{attribute addProperty BoxType "EL6851-0010-0019"}
{attribute addProperty Id "DMX_StatusAT %I*DMX_Status_A8F3522A6480DMX_Channel_1_64AT %I*DMX_Channel_D03720FB512640WcStateAT %I*WcState_98A4DF7520.250InfoDataAT %I*InfoData_BC63D37F80100"}
{attribute addProperty CRC "2912125561"}
{attribute addProperty SizeInBites "658"}
{attribute addProperty SizeInBytes "82.25"}
TYPE EL6851_20762A18 :
STRUCT
	{attribute addProperty Name "DMX_Status"}
	DMX_Status : DMX_Status_A8F3522A;
	{attribute addProperty Name "DMX_Channel_1_64"}
	DMX_Channel_1_64 : DMX_Channel_D03720FB;
	{attribute addProperty Name "WcState"}
	WcState : WcState_98A4DF75;
	{attribute addProperty Name "InfoData"}
	InfoData : InfoData_BC63D37F;
END_STRUCT
END_TYPE

(* stored: Version 1.2.0.0, ProductVersion 3.1.4024.9
   DUT EL6851_20762A18: Id {6cf03f40-00a6-40c4-97e8-d86fc01b4f43} *)
